FUNCTION_BLOCK CoverIO EXTENDS SM_CoverIO
VAR_INPUT
END_VAR
VAR_OUTPUT
END_VAR
VAR
    _testVar : INT;
END_VAR

SUPER^();

// do stuff

//SUPER^();

END_FUNCTION_BLOCK

(* stored: Version 1.1.0.1, ProductVersion 3.1.4018.2
   POU CoverIO: Id {7179e359-56e0-423b-b637-b5905b503c88}, SpecialFunc None *)
